FUNCTION_BLOCK 2D_MOVETO_XY_COORD (* Move to location keeping 'z' constant *)
  (* Standard: 61499-2 *)
  (* Version 26-03-12, GASR *)
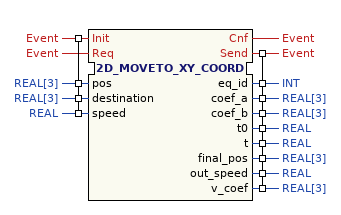
  EVENT_INPUT
    Init WITH pos, destination, speed; (* Initialization Request *)
    Req; (* Requisition to finish *)
  END_EVENT
  EVENT_OUTPUT
    Cnf; (* Execution confirmed *)
    Send WITH eq_id, coef_a, coef_b, t0, t, final_pos, out_speed, v_coef; (* Send data to output *)
  END_EVENT
  VAR_INPUT
    pos : ARRAY [0..2] OF REAL; (* Machine position *)
    destination : ARRAY [0..2] OF REAL;
    speed : REAL := 0; (* Speed in m/s *)
  END_VAR
  VAR_OUTPUT
    eq_id : INT; (* Curve equation type id *)
    coef_a : ARRAY [0..2] OF REAL; (* Line angular coeficients *)
    coef_b : ARRAY [0..2] OF REAL; (* Line linear coeficients *)
    t0 : REAL; (* Initial parameter *)
    t : REAL; (* Final parameter *)
    final_pos : ARRAY [0..2] OF REAL; (* Final position *)
    out_speed : REAL; (* Speed in m/s *)
    v_coef : ARRAY [0..2] OF REAL; (* Velocity coeficients *)
  END_VAR
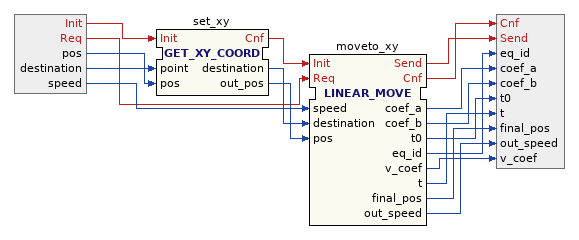
  FBS
    set_xy : GET_XY_COORD;
    moveto_xy : LINEAR_MOVE;
  END_FBS
  EVENT_CONNECTIONS
    set_xy.Cnf TO moveto_xy.Init;
    moveto_xy.Send TO Send;
    moveto_xy.Cnf TO Cnf;
    Init TO set_xy.Init;
    Req TO moveto_xy.Req;
  END_CONNECTIONS
  DATA_CONNECTIONS
    speed TO moveto_xy.speed;
    set_xy.destination TO moveto_xy.destination;
    set_xy.out_pos TO moveto_xy.pos;
    destination TO set_xy.point;
    pos TO set_xy.pos;
    moveto_xy.coef_a TO coef_a;
    moveto_xy.coef_b TO coef_b;
    moveto_xy.t0 TO t0;
    moveto_xy.eq_id TO eq_id;
    moveto_xy.v_coef TO v_coef;
    moveto_xy.t TO t;
    moveto_xy.final_pos TO final_pos;
    moveto_xy.out_speed TO out_speed;
  END_CONNECTIONS
END_FUNCTION_BLOCK
